PROGRAM MAIN
VAR
	fbIntersection : FB_Intersection;
    tonAdvance     : TON;                        // timer between phase advances
    PHASE_TIME     : TIME := T#5S;               // how long each phase lasts
	bManualAdvance : BOOL := FALSE;			     // HMI button
END_VAR

// Auto-advance on timer
tonAdvance(IN := NOT tonAdvance.Q, PT := PHASE_TIME);
IF (tonAdvance.Q) THEN
    fbIntersection.Advance();
END_IF

// Manual advance from HMI (edge-detected inside the intersection)
fbIntersection.Update(bManualStepRequest := bManualAdvance);
bManualAdvance := FALSE;

END_PROGRAM

(* stored: Version 1.1.0.1, ProductVersion 3.1.4024.12
   POU MAIN: Id {7d9e93e5-9bb5-44fa-aa35-8d8935fc199d}, SpecialFunc None *)
